// Mitsubishi GX Developer project: Китай гильотина   PLC: FX3U

PROGRAM MAIN
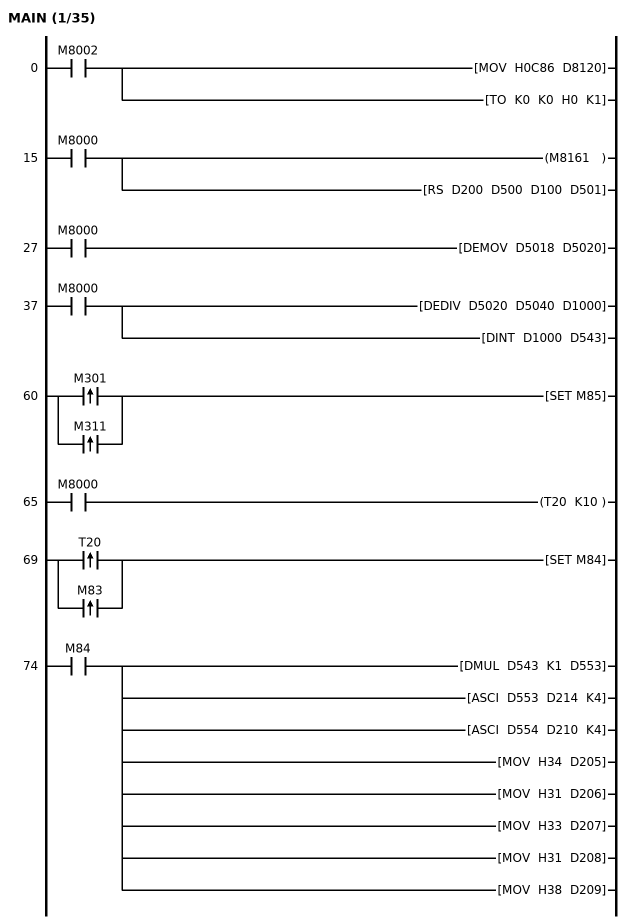
0     LD      M8002
      MOV     H0C86 D8120
      TO      K0 K0 H0 K1
15    LD      M8000
      OUT     M8161
      RS      D200 D500 D100 D501
27    LD      M8000
      DEMOV   D5018 D5020
37    LD      M8000
      DEDIV   D5020 D5040 D1000
      DINT    D1000 D543
60    LDP     M301
      ORP     M311
      SET     M85
65    LD      M8000
      OUT     T20 K10
69    LDP     T20
      ORP     M83
      SET     M84
74    LD      M84
      DMUL    D543 K1 D553
      ASCI    D553 D214 K4
      ASCI    D554 D210 K4
      MOV     H34 D205
      MOV     H31 D206
      MOV     H33 D207
      MOV     H31 D208
      MOV     H38 D209
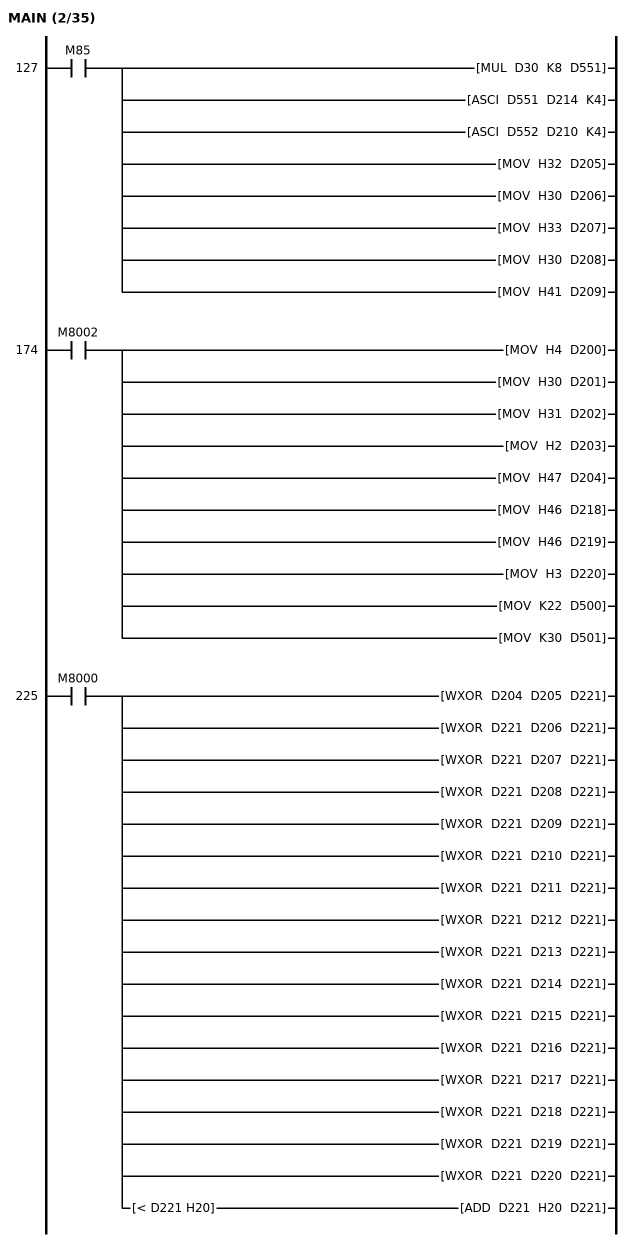
127   LD      M85
      MUL     D30 K8 D551
      ASCI    D551 D214 K4
      ASCI    D552 D210 K4
      MOV     H32 D205
      MOV     H30 D206
      MOV     H33 D207
      MOV     H30 D208
      MOV     H41 D209
174   LD      M8002
      MOV     H4 D200
      MOV     H30 D201
      MOV     H31 D202
      MOV     H2 D203
      MOV     H47 D204
      MOV     H46 D218
      MOV     H46 D219
      MOV     H3 D220
      MOV     K22 D500
      MOV     K30 D501
225   LD      M8000
      WXOR    D204 D205 D221
      WXOR    D221 D206 D221
      WXOR    D221 D207 D221
      WXOR    D221 D208 D221
      WXOR    D221 D209 D221
      WXOR    D221 D210 D221
      WXOR    D221 D211 D221
      WXOR    D221 D212 D221
      WXOR    D221 D213 D221
      WXOR    D221 D214 D221
      WXOR    D221 D215 D221
      WXOR    D221 D216 D221
      WXOR    D221 D217 D221
      WXOR    D221 D218 D221
      WXOR    D221 D219 D221
      WXOR    D221 D220 D221
      AND<    D221 H20
      ADD     D221 H20 D221
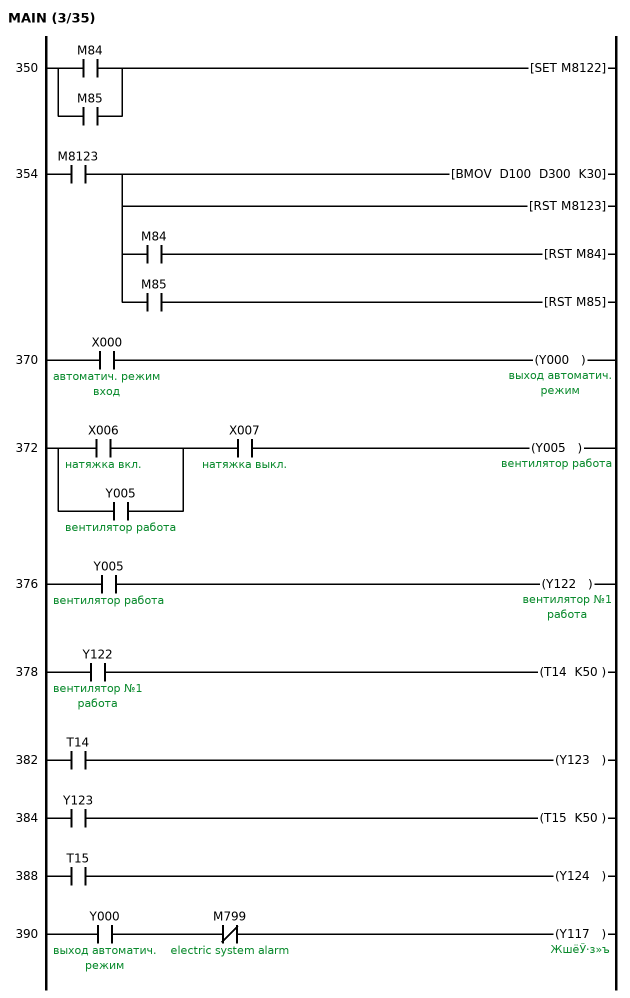
350   LD      M84
      OR      M85
      SET     M8122
354   LD      M8123
      BMOV    D100 D300 K30
      RST     M8123
      MPS
      AND     M84
      RST     M84
      MPP
      AND     M85
      RST     M85
370   LD      X000  ; автоматич. режим вход
      OUT     Y000  ; выход автоматич. режим
372   LD      X006  ; натяжка вкл.
      OR      Y005  ; вентилятор работа
      AND     X007  ; натяжка выкл.
      OUT     Y005  ; вентилятор работа
376   LD      Y005  ; вентилятор работа
      OUT     Y122  ; вентилятор №1 работа
378   LD      Y122  ; вентилятор №1 работа
      OUT     T14 K50
382   LD      T14
      OUT     Y123
384   LD      Y123
      OUT     T15 K50
388   LD      T15
      OUT     Y124
390   LD      Y000  ; выход автоматич. режим
      ANI     M799  ; electric system alarm
      OUT     Y117  ; ЖшёЎ·з»ъ
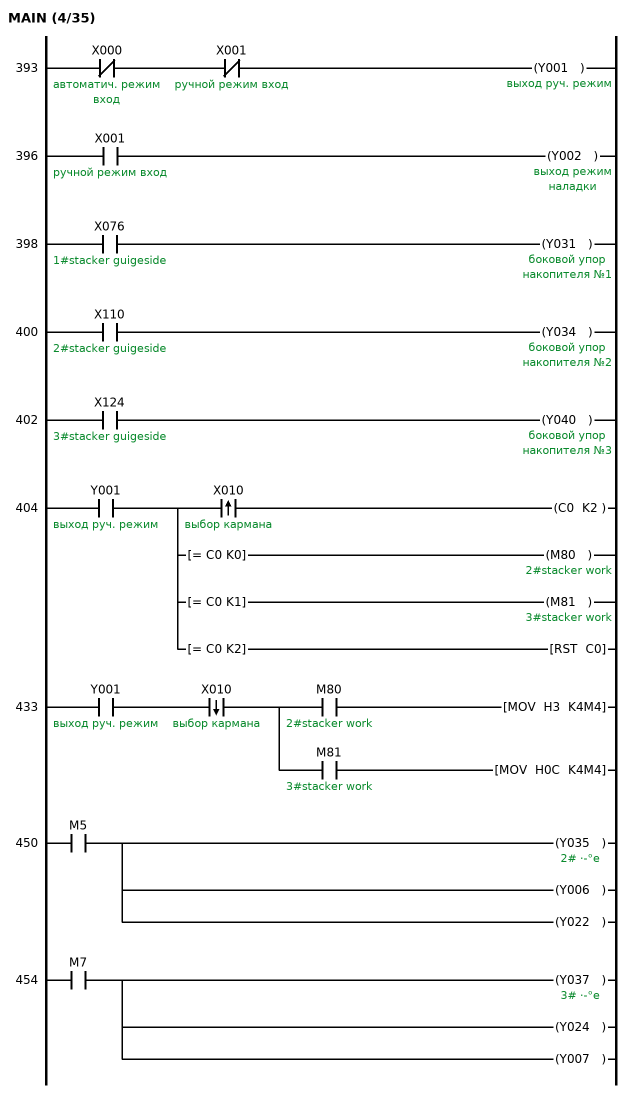
393   LDI     X000  ; автоматич. режим вход
      ANI     X001  ; ручной режим вход
      OUT     Y001  ; выход руч. режим
396   LD      X001  ; ручной режим вход
      OUT     Y002  ; выход режим наладки
398   LD      X076  ; 1#stacker guigeside
      OUT     Y031  ; боковой упор накопителя №1
400   LD      X110  ; 2#stacker guigeside
      OUT     Y034  ; боковой упор накопителя №2
402   LD      X124  ; 3#stacker guigeside
      OUT     Y040  ; боковой упор накопителя №3
404   LD      Y001  ; выход руч. режим
      MPS
      ANDP    X010  ; выбор кармана
      OUT     C0 K2
      MRD
      AND=    C0 K0
      OUT     M80  ; 2#stacker work
      MRD
      AND=    C0 K1
      OUT     M81  ; 3#stacker work
      MPP
      AND=    C0 K2
      RST     C0
433   LD      Y001  ; выход руч. режим
      ANDF    X010  ; выбор кармана
      MPS
      AND     M80  ; 2#stacker work
      MOV     H3 K4M4
      MPP
      AND     M81  ; 3#stacker work
      MOV     H0C K4M4
450   LD      M5
      OUT     Y035  ; 2# ·­°е
      OUT     Y006
      OUT     Y022
454   LD      M7
      OUT     Y037  ; 3# ·­°е
      OUT     Y024
      OUT     Y007
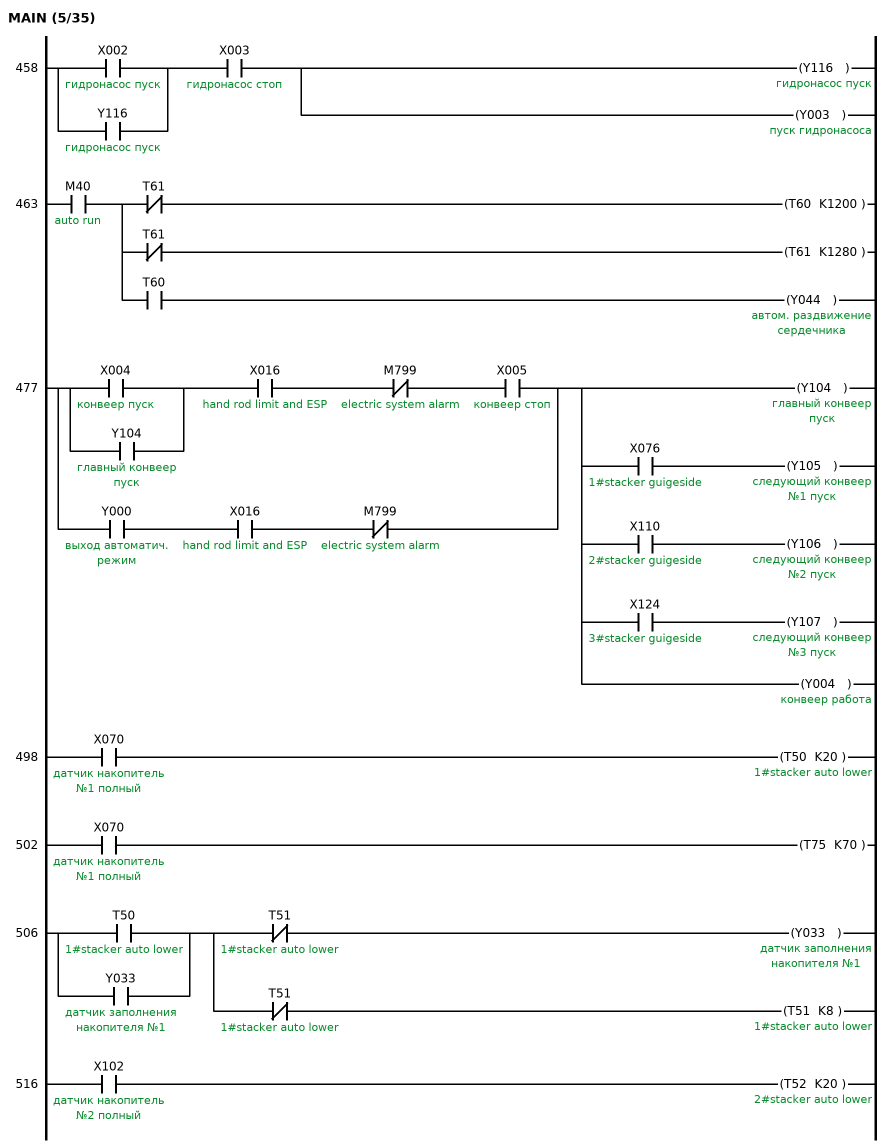
458   LD      X002  ; гидронасос пуск
      OR      Y116  ; гидронасос пуск
      AND     X003  ; гидронасос стоп
      OUT     Y116  ; гидронасос пуск
      OUT     Y003  ; пуск гидронасоса
463   LD      M40  ; auto run
      MPS
      ANI     T61
      OUT     T60 K1200
      MRD
      ANI     T61
      OUT     T61 K1280
      MPP
      AND     T60
      OUT     Y044  ; автом. раздвижение сердечника
477   LD      X004  ; конвеер пуск
      OR      Y104  ; главный конвеер пуск
      AND     X016  ; hand rod limit and ESP
      ANI     M799  ; electric system alarm
      AND     X005  ; конвеер стоп
      LD      Y000  ; выход автоматич. режим
      AND     X016  ; hand rod limit and ESP
      ANI     M799  ; electric system alarm
      ORB
      OUT     Y104  ; главный конвеер пуск
      MPS
      AND     X076  ; 1#stacker guigeside
      OUT     Y105  ; следующий конвеер №1 пуск
      MRD
      AND     X110  ; 2#stacker guigeside
      OUT     Y106  ; следующий конвеер №2 пуск
      MRD
      AND     X124  ; 3#stacker guigeside
      OUT     Y107  ; следующий конвеер №3 пуск
      MPP
      OUT     Y004  ; конвеер работа
498   LD      X070  ; датчик накопитель №1 полный
      OUT     T50 K20  ; 1#stacker auto lower
502   LD      X070  ; датчик накопитель №1 полный
      OUT     T75 K70
506   LD      T50  ; 1#stacker auto lower
      OR      Y033  ; датчик заполнения накопителя №1
      MPS
      ANI     T51  ; 1#stacker auto lower
      OUT     Y033  ; датчик заполнения накопителя №1
      MPP
      ANI     T51  ; 1#stacker auto lower
      OUT     T51 K8  ; 1#stacker auto lower
516   LD      X102  ; датчик накопитель №2 полный
      OUT     T52 K20  ; 2#stacker auto lower
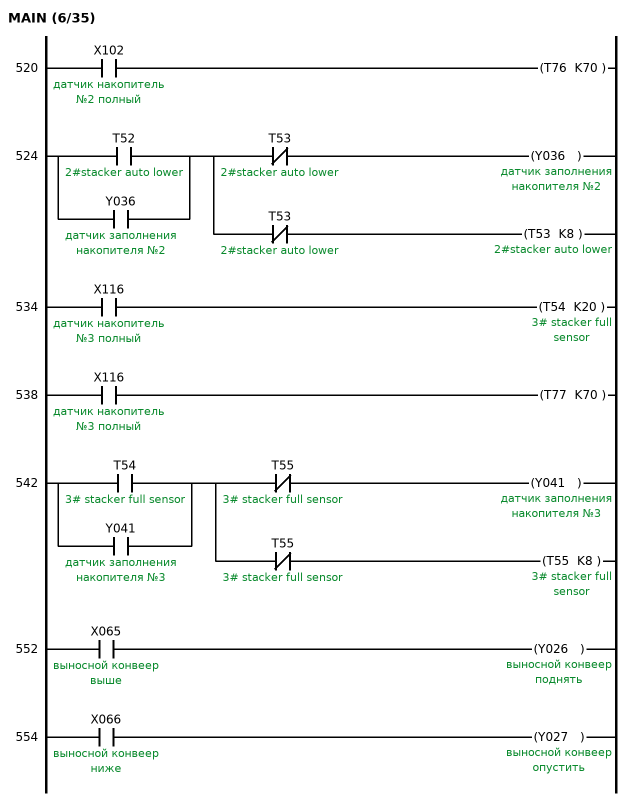
520   LD      X102  ; датчик накопитель №2 полный
      OUT     T76 K70
524   LD      T52  ; 2#stacker auto lower
      OR      Y036  ; датчик заполнения накопителя №2
      MPS
      ANI     T53  ; 2#stacker auto lower
      OUT     Y036  ; датчик заполнения накопителя №2
      MPP
      ANI     T53  ; 2#stacker auto lower
      OUT     T53 K8  ; 2#stacker auto lower
534   LD      X116  ; датчик накопитель №3 полный
      OUT     T54 K20  ; 3# stacker full sensor
538   LD      X116  ; датчик накопитель №3 полный
      OUT     T77 K70
542   LD      T54  ; 3# stacker full sensor
      OR      Y041  ; датчик заполнения накопителя №3
      MPS
      ANI     T55  ; 3# stacker full sensor
      OUT     Y041  ; датчик заполнения накопителя №3
      MPP
      ANI     T55  ; 3# stacker full sensor
      OUT     T55 K8  ; 3# stacker full sensor
552   LD      X065  ; выносной конвеер выше
      OUT     Y026  ; выносной конвеер поднять
554   LD      X066  ; выносной конвеер ниже
      OUT     Y027  ; выносной конвеер опустить
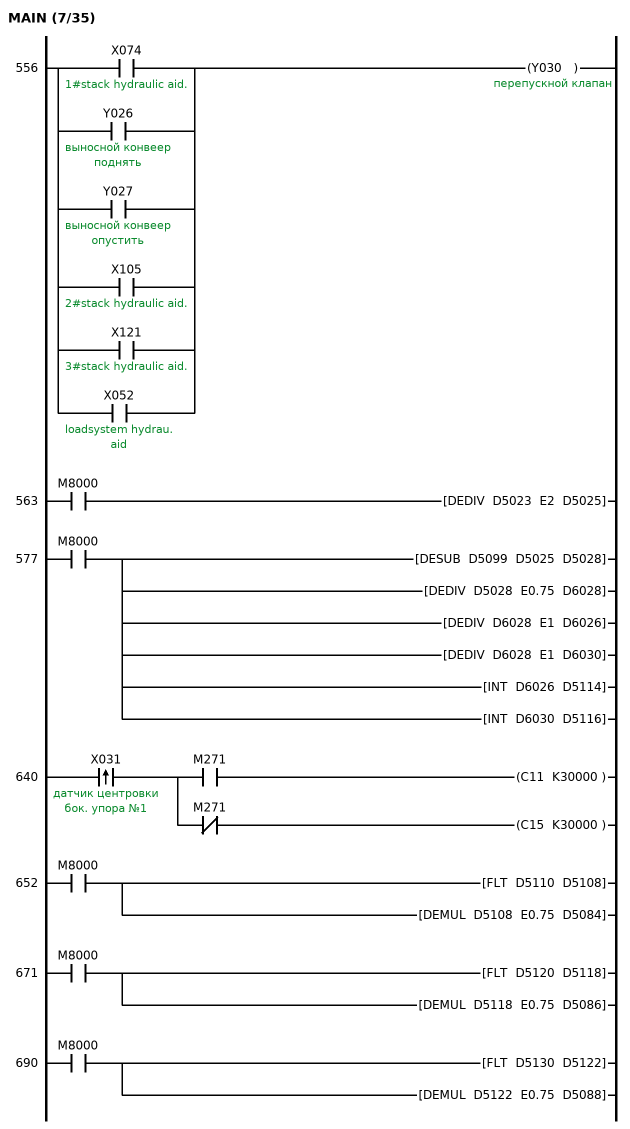
556   LD      X074  ; 1#stack hydraulic aid.
      OR      Y026  ; выносной конвеер поднять
      OR      Y027  ; выносной конвеер опустить
      OR      X105  ; 2#stack hydraulic aid.
      OR      X121  ; 3#stack hydraulic aid.
      OR      X052  ; loadsystem hydrau. aid
      OUT     Y030  ; перепускной клапан
563   LD      M8000
      DEDIV   D5023 E2 D5025
577   LD      M8000
      DESUB   D5099 D5025 D5028
      DEDIV   D5028 E0.75 D6028
      DEDIV   D6028 E1 D6026
      DEDIV   D6028 E1 D6030
      INT     D6026 D5114
      INT     D6030 D5116
640   LDP     X031  ; датчик центровки бок. упора №1
      MPS
      AND     M271
      OUT     C11 K30000
      MPP
      ANI     M271
      OUT     C15 K30000
652   LD      M8000
      FLT     D5110 D5108
      DEMUL   D5108 E0.75 D5084
671   LD      M8000
      FLT     D5120 D5118
      DEMUL   D5118 E0.75 D5086
690   LD      M8000
      FLT     D5130 D5122
      DEMUL   D5122 E0.75 D5088
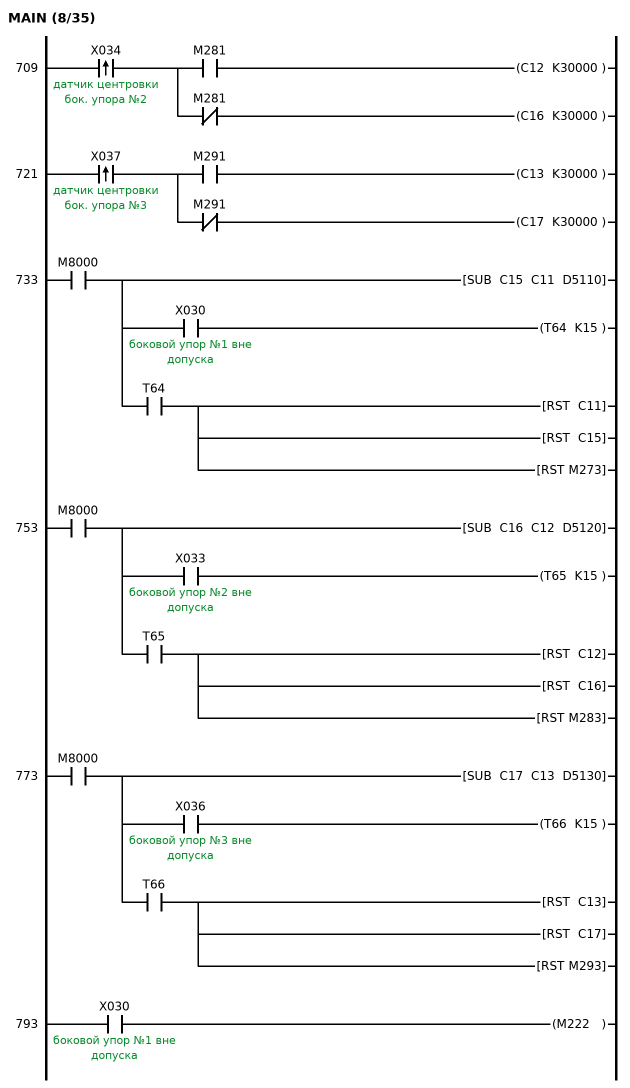
709   LDP     X034  ; датчик центровки бок. упора №2
      MPS
      AND     M281
      OUT     C12 K30000
      MPP
      ANI     M281
      OUT     C16 K30000
721   LDP     X037  ; датчик центровки бок. упора №3
      MPS
      AND     M291
      OUT     C13 K30000
      MPP
      ANI     M291
      OUT     C17 K30000
733   LD      M8000
      SUB     C15 C11 D5110
      MPS
      AND     X030  ; боковой упор №1 вне допуска
      OUT     T64 K15
      MPP
      AND     T64
      RST     C11
      RST     C15
      RST     M273
753   LD      M8000
      SUB     C16 C12 D5120
      MPS
      AND     X033  ; боковой упор №2 вне допуска
      OUT     T65 K15
      MPP
      AND     T65
      RST     C12
      RST     C16
      RST     M283
773   LD      M8000
      SUB     C17 C13 D5130
      MPS
      AND     X036  ; боковой упор №3 вне допуска
      OUT     T66 K15
      MPP
      AND     T66
      RST     C13
      RST     C17
      RST     M293
793   LD      X030  ; боковой упор №1 вне допуска
      OUT     M222
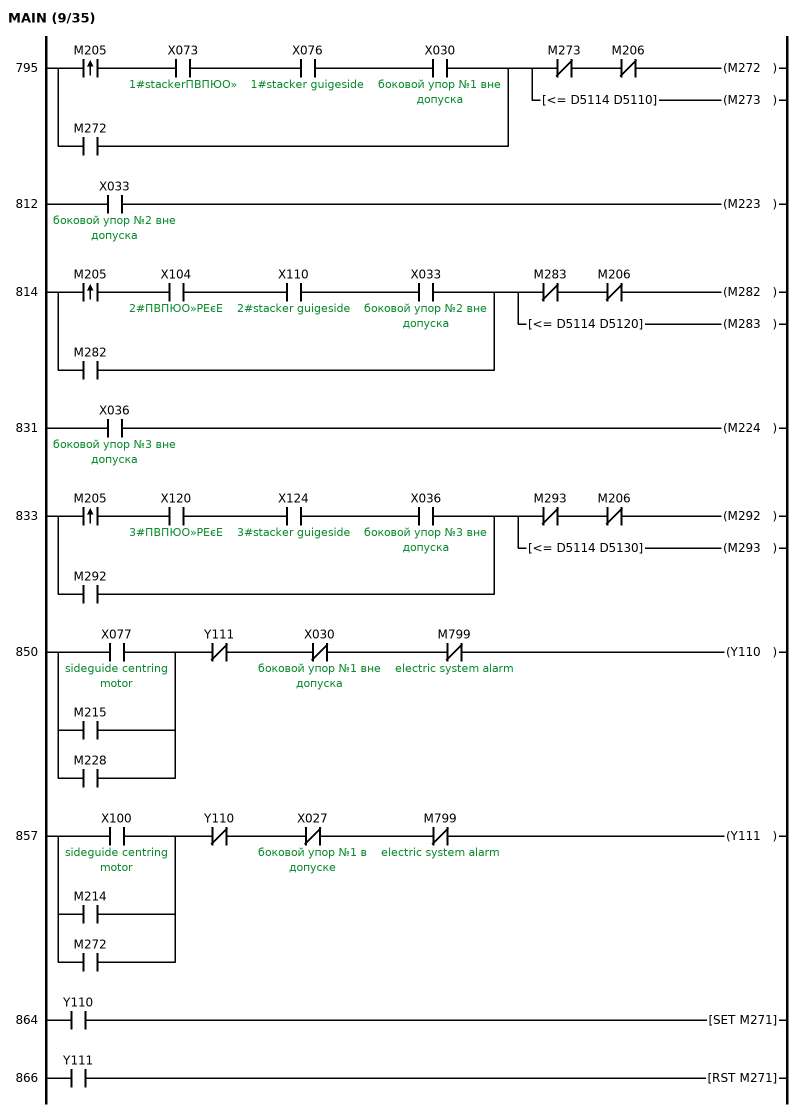
795   LDP     M205
      AND     X073  ; 1#stackerПВПЮО»
      AND     X076  ; 1#stacker guigeside
      AND     X030  ; боковой упор №1 вне допуска
      OR      M272
      MPS
      ANI     M273
      ANI     M206
      OUT     M272
      MPP
      AND<=   D5114 D5110
      OUT     M273
812   LD      X033  ; боковой упор №2 вне допуска
      OUT     M223
814   LDP     M205
      AND     X104  ; 2#ПВПЮО»РЕєЕ
      AND     X110  ; 2#stacker guigeside
      AND     X033  ; боковой упор №2 вне допуска
      OR      M282
      MPS
      ANI     M283
      ANI     M206
      OUT     M282
      MPP
      AND<=   D5114 D5120
      OUT     M283
831   LD      X036  ; боковой упор №3 вне допуска
      OUT     M224
833   LDP     M205
      AND     X120  ; 3#ПВПЮО»РЕєЕ
      AND     X124  ; 3#stacker guigeside
      AND     X036  ; боковой упор №3 вне допуска
      OR      M292
      MPS
      ANI     M293
      ANI     M206
      OUT     M292
      MPP
      AND<=   D5114 D5130
      OUT     M293
850   LD      X077  ; sideguide centring motor
      OR      M215
      OR      M228
      ANI     Y111
      ANI     X030  ; боковой упор №1 вне допуска
      ANI     M799  ; electric system alarm
      OUT     Y110
857   LD      X100  ; sideguide centring motor
      OR      M214
      OR      M272
      ANI     Y110
      ANI     X027  ; боковой упор №1 в допуске
      ANI     M799  ; electric system alarm
      OUT     Y111
864   LD      Y110
      SET     M271
866   LD      Y111
      RST     M271
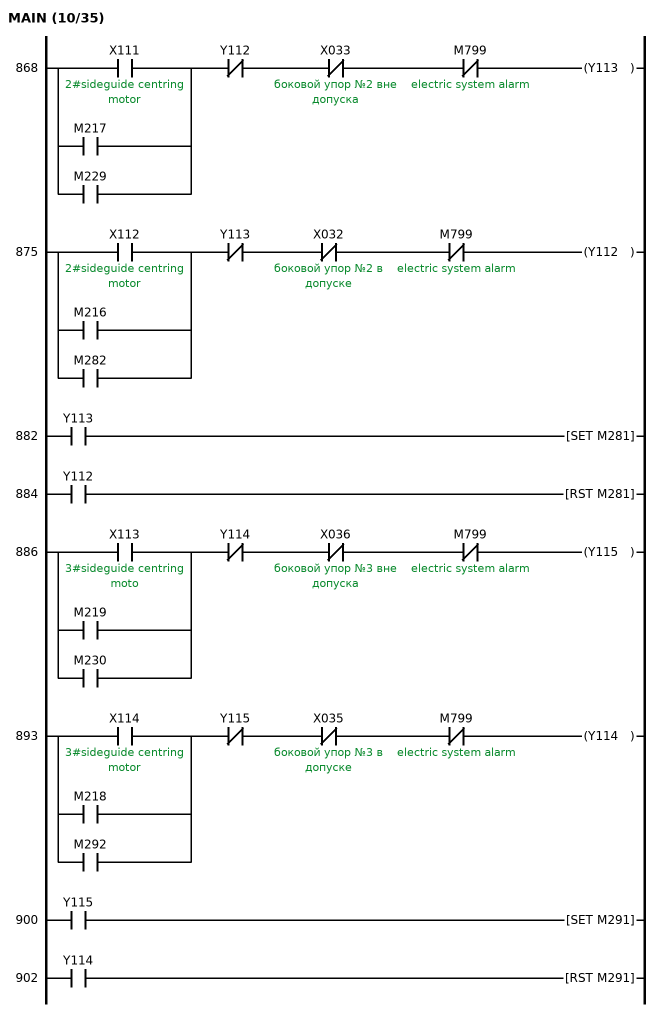
868   LD      X111  ; 2#sideguide centring motor
      OR      M217
      OR      M229
      ANI     Y112
      ANI     X033  ; боковой упор №2 вне допуска
      ANI     M799  ; electric system alarm
      OUT     Y113
875   LD      X112  ; 2#sideguide centring motor
      OR      M216
      OR      M282
      ANI     Y113
      ANI     X032  ; боковой упор №2 в допуске
      ANI     M799  ; electric system alarm
      OUT     Y112
882   LD      Y113
      SET     M281
884   LD      Y112
      RST     M281
886   LD      X113  ; 3#sideguide centring moto
      OR      M219
      OR      M230
      ANI     Y114
      ANI     X036  ; боковой упор №3 вне допуска
      ANI     M799  ; electric system alarm
      OUT     Y115
893   LD      X114  ; 3#sideguide centring motor
      OR      M218
      OR      M292
      ANI     Y115
      ANI     X035  ; боковой упор №3 в допуске
      ANI     M799  ; electric system alarm
      OUT     Y114
900   LD      Y115
      SET     M291
902   LD      Y114
      RST     M291
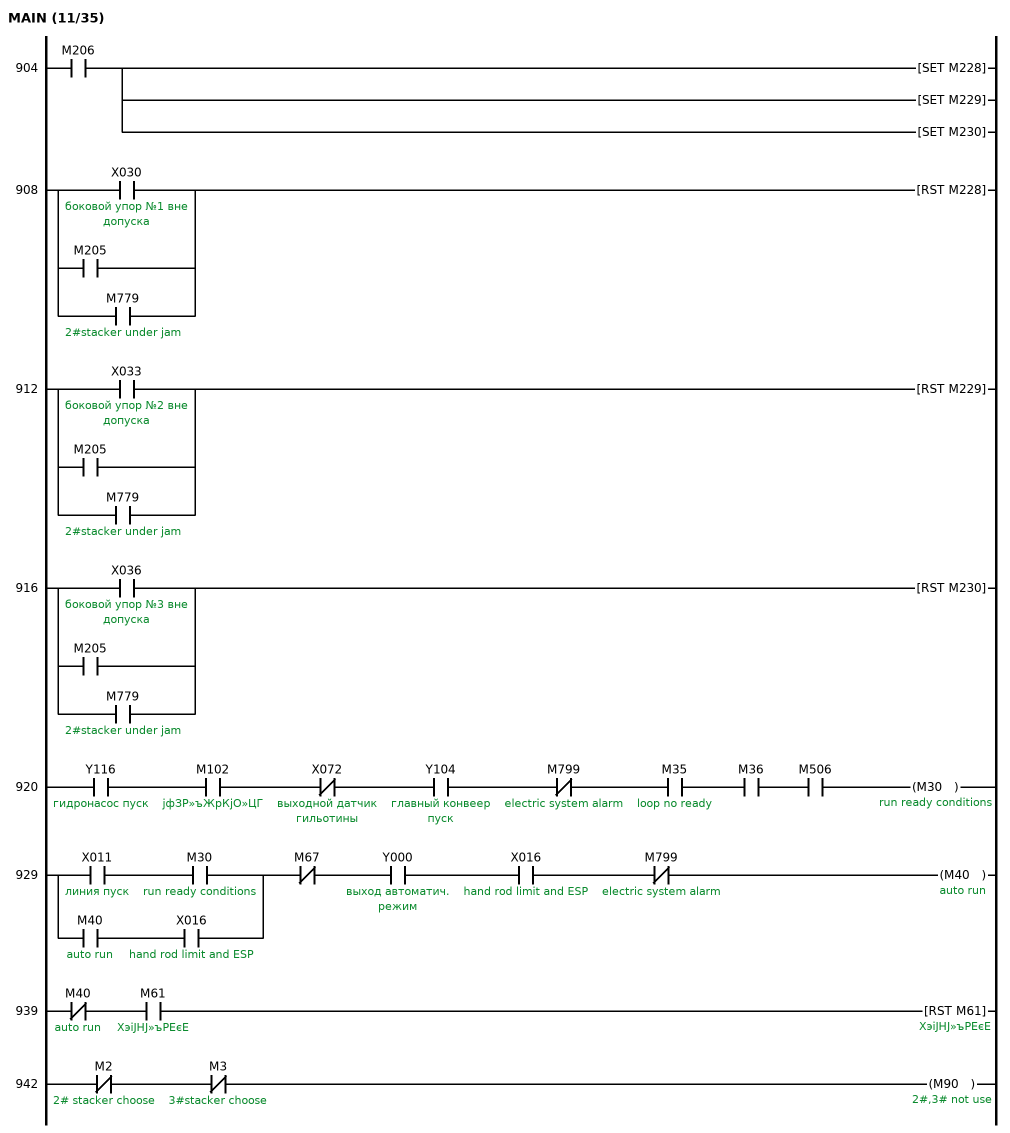
904   LD      M206
      SET     M228
      SET     M229
      SET     M230
908   LD      X030  ; боковой упор №1 вне допуска
      OR      M205
      OR      M779  ; 2#stacker under jam
      RST     M228
912   LD      X033  ; боковой упор №2 вне допуска
      OR      M205
      OR      M779  ; 2#stacker under jam
      RST     M229
916   LD      X036  ; боковой упор №3 вне допуска
      OR      M205
      OR      M779  ; 2#stacker under jam
      RST     M230
920   LD      Y116  ; гидронасос пуск
      AND     M102  ; јфЗР»ъЖрКјО»ЦГ
      ANI     X072  ; выходной датчик гильотины
      AND     Y104  ; главный конвеер пуск
      ANI     M799  ; electric system alarm
      AND     M35  ; loop no ready
      AND     M36
      AND     M506
      OUT     M30  ; run ready conditions
929   LD      X011  ; линия пуск
      AND     M30  ; run ready conditions
      LD      M40  ; auto run
      AND     X016  ; hand rod limit and ESP
      ORB
      ANI     M67
      AND     Y000  ; выход автоматич. режим
      AND     X016  ; hand rod limit and ESP
      ANI     M799  ; electric system alarm
      OUT     M40  ; auto run
939   LDI     M40  ; auto run
      AND     M61  ; ХэіЈНЈ»ъРЕєЕ
      RST     M61  ; ХэіЈНЈ»ъРЕєЕ
942   LDI     M2  ; 2# stacker choose
      ANI     M3  ; 3#stacker choose
      OUT     M90  ; 2#,3# not use
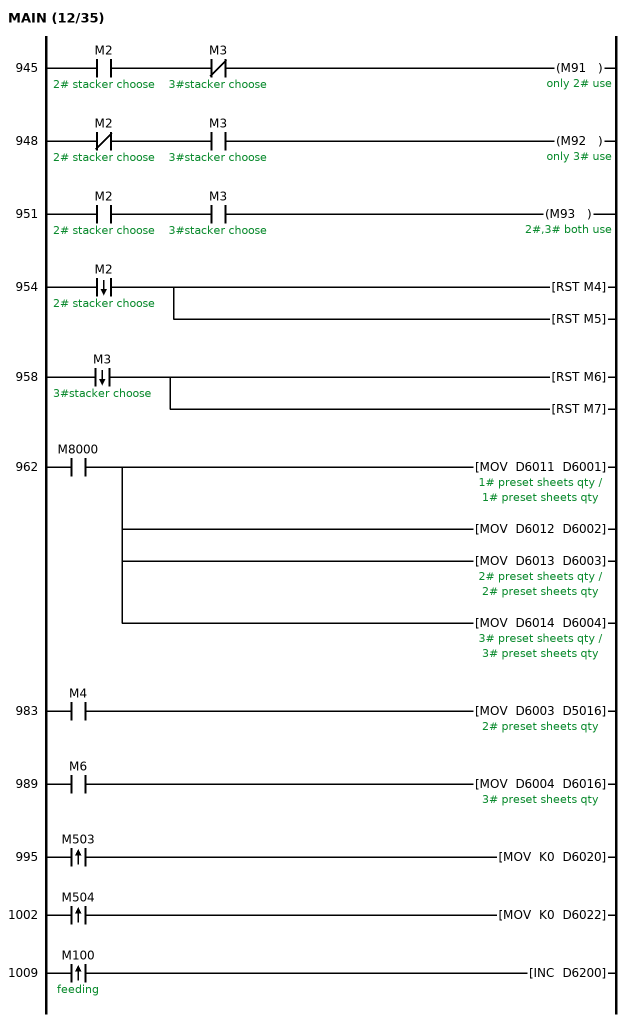
945   LD      M2  ; 2# stacker choose
      ANI     M3  ; 3#stacker choose
      OUT     M91  ; only 2# use
948   LDI     M2  ; 2# stacker choose
      AND     M3  ; 3#stacker choose
      OUT     M92  ; only 3# use
951   LD      M2  ; 2# stacker choose
      AND     M3  ; 3#stacker choose
      OUT     M93  ; 2#,3# both use
954   LDF     M2  ; 2# stacker choose
      RST     M4
      RST     M5
958   LDF     M3  ; 3#stacker choose
      RST     M6
      RST     M7
962   LD      M8000
      MOV     D6011 D6001  ; 1# preset sheets qty / 1# preset sheets qty
      MOV     D6012 D6002
      MOV     D6013 D6003  ; 2# preset sheets qty / 2# preset sheets qty
      MOV     D6014 D6004  ; 3# preset sheets qty / 3# preset sheets qty
983   LD      M4
      MOV     D6003 D5016
989   LD      M6
      MOV     D6004 D6016
995   LDP     M503
      MOV     K0 D6020
1002  LDP     M504
      MOV     K0 D6022
1009  LDP     M100  ; feeding
      INC     D6200
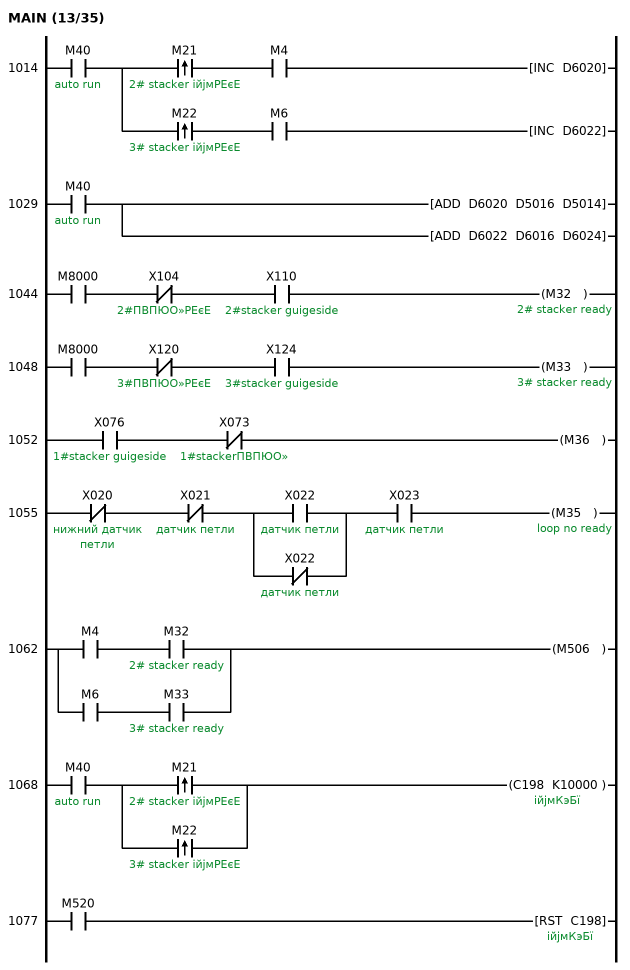
1014  LD      M40  ; auto run
      MPS
      ANDP    M21  ; 2# stacker ійјмРЕєЕ
      AND     M4
      INC     D6020
      MPP
      ANDP    M22  ; 3# stacker ійјмРЕєЕ
      AND     M6
      INC     D6022
1029  LD      M40  ; auto run
      ADD     D6020 D5016 D5014
      ADD     D6022 D6016 D6024
1044  LD      M8000
      ANI     X104  ; 2#ПВПЮО»РЕєЕ
      AND     X110  ; 2#stacker guigeside
      OUT     M32  ; 2# stacker ready
1048  LD      M8000
      ANI     X120  ; 3#ПВПЮО»РЕєЕ
      AND     X124  ; 3#stacker guigeside
      OUT     M33  ; 3# stacker ready
1052  LD      X076  ; 1#stacker guigeside
      ANI     X073  ; 1#stackerПВПЮО»
      OUT     M36
1055  LDI     X020  ; нижний датчик петли
      ANI     X021  ; датчик петли
      LD      X022  ; датчик петли
      ORI     X022  ; датчик петли
      ANB
      AND     X023  ; датчик петли
      OUT     M35  ; loop no ready
1062  LD      M4
      AND     M32  ; 2# stacker ready
      LD      M6
      AND     M33  ; 3# stacker ready
      ORB
      OUT     M506
1068  LD      M40  ; auto run
      LDP     M21  ; 2# stacker ійјмРЕєЕ
      ORP     M22  ; 3# stacker ійјмРЕєЕ
      ANB
      OUT     C198 K10000  ; ійјмКэБї
1077  LD      M520
      RST     C198  ; ійјмКэБї
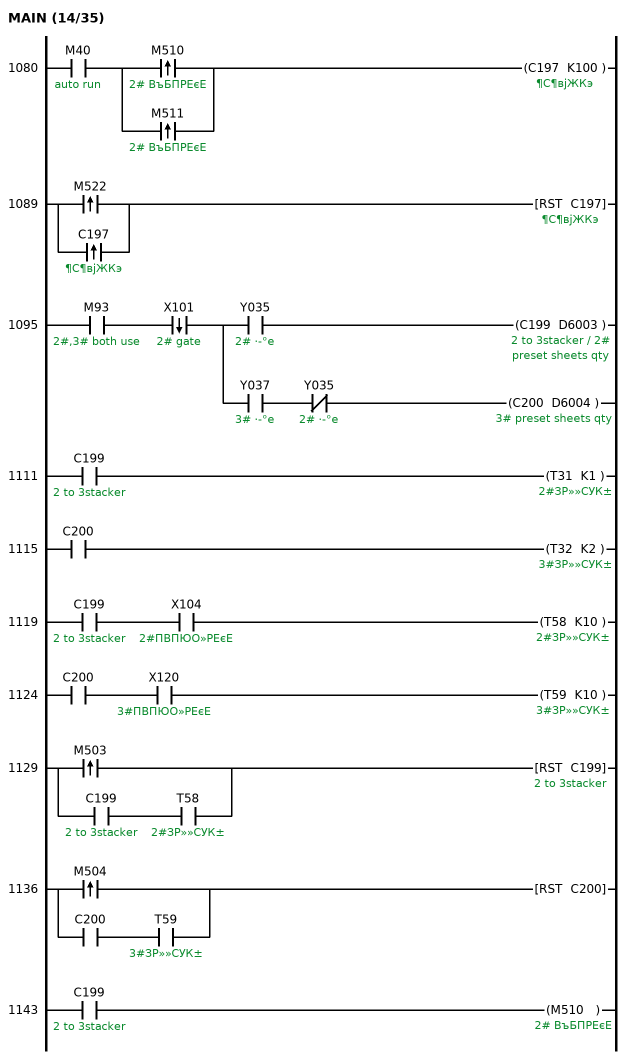
1080  LD      M40  ; auto run
      LDP     M510  ; 2# ВъБПРЕєЕ
      ORP     M511  ; 2# ВъБПРЕєЕ
      ANB
      OUT     C197 K100  ; ¶С¶вјЖКэ
1089  LDP     M522
      ORP     C197  ; ¶С¶вјЖКэ
      RST     C197  ; ¶С¶вјЖКэ
1095  LD      M93  ; 2#,3# both use
      ANDF    X101  ; 2# gate
      MPS
      AND     Y035  ; 2# ·­°е
      OUT     C199 D6003  ; 2 to 3stacker / 2# preset sheets qty
      MPP
      AND     Y037  ; 3# ·­°е
      ANI     Y035  ; 2# ·­°е
      OUT     C200 D6004  ; 3# preset sheets qty
1111  LD      C199  ; 2 to 3stacker
      OUT     T31 K1  ; 2#ЗР»»СУК±
1115  LD      C200
      OUT     T32 K2  ; 3#ЗР»»СУК±
1119  LD      C199  ; 2 to 3stacker
      AND     X104  ; 2#ПВПЮО»РЕєЕ
      OUT     T58 K10  ; 2#ЗР»»СУК±
1124  LD      C200
      AND     X120  ; 3#ПВПЮО»РЕєЕ
      OUT     T59 K10  ; 3#ЗР»»СУК±
1129  LDP     M503
      LD      C199  ; 2 to 3stacker
      AND     T58  ; 2#ЗР»»СУК±
      ORB
      RST     C199  ; 2 to 3stacker
1136  LDP     M504
      LD      C200
      AND     T59  ; 3#ЗР»»СУК±
      ORB
      RST     C200
1143  LD      C199  ; 2 to 3stacker
      OUT     M510  ; 2# ВъБПРЕєЕ
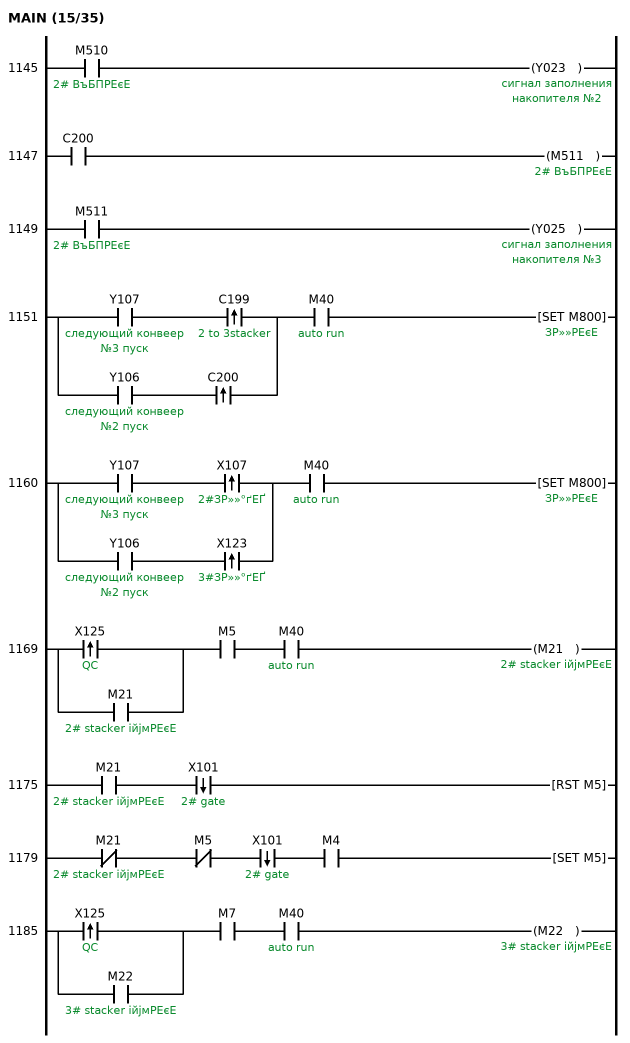
1145  LD      M510  ; 2# ВъБПРЕєЕ
      OUT     Y023  ; сигнал заполнения накопителя №2
1147  LD      C200
      OUT     M511  ; 2# ВъБПРЕєЕ
1149  LD      M511  ; 2# ВъБПРЕєЕ
      OUT     Y025  ; сигнал заполнения накопителя №3
1151  LD      Y107  ; следующий конвеер №3 пуск
      ANDP    C199  ; 2 to 3stacker
      LD      Y106  ; следующий конвеер №2 пуск
      ANDP    C200
      ORB
      AND     M40  ; auto run
      SET     M800  ; ЗР»»РЕєЕ
1160  LD      Y107  ; следующий конвеер №3 пуск
      ANDP    X107  ; 2#ЗР»»°ґЕҐ
      LD      Y106  ; следующий конвеер №2 пуск
      ANDP    X123  ; 3#ЗР»»°ґЕҐ
      ORB
      AND     M40  ; auto run
      SET     M800  ; ЗР»»РЕєЕ
1169  LDP     X125  ; QC
      OR      M21  ; 2# stacker ійјмРЕєЕ
      AND     M5
      AND     M40  ; auto run
      OUT     M21  ; 2# stacker ійјмРЕєЕ
1175  LD      M21  ; 2# stacker ійјмРЕєЕ
      ANDF    X101  ; 2# gate
      RST     M5
1179  LDI     M21  ; 2# stacker ійјмРЕєЕ
      ANI     M5
      ANDF    X101  ; 2# gate
      AND     M4
      SET     M5
1185  LDP     X125  ; QC
      OR      M22  ; 3# stacker ійјмРЕєЕ
      AND     M7
      AND     M40  ; auto run
      OUT     M22  ; 3# stacker ійјмРЕєЕ
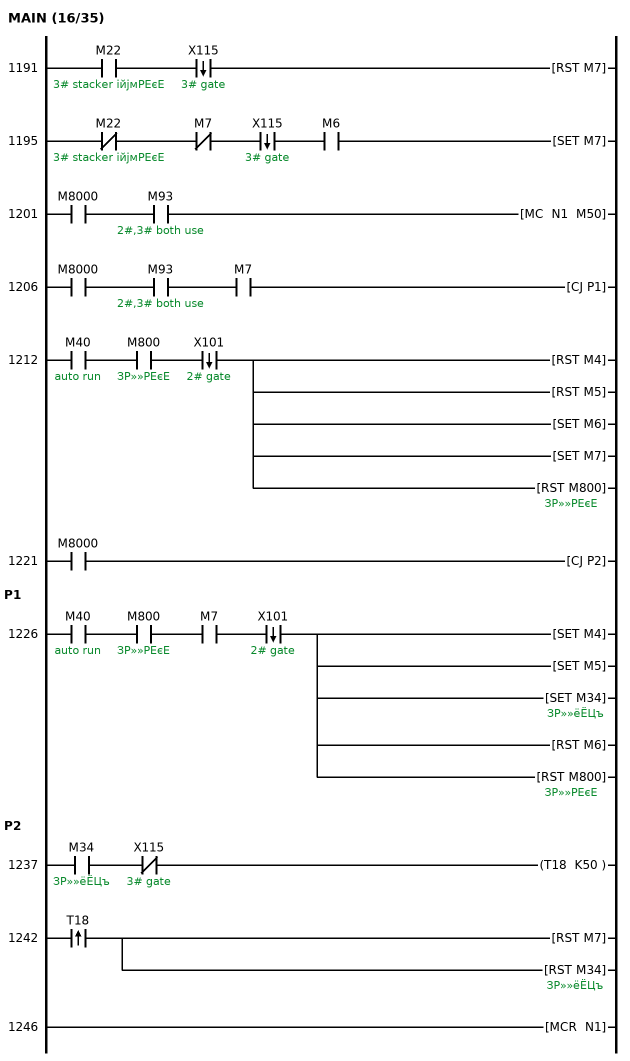
1191  LD      M22  ; 3# stacker ійјмРЕєЕ
      ANDF    X115  ; 3# gate
      RST     M7
1195  LDI     M22  ; 3# stacker ійјмРЕєЕ
      ANI     M7
      ANDF    X115  ; 3# gate
      AND     M6
      SET     M7
1201  LD      M8000
      AND     M93  ; 2#,3# both use
      MC      N1 M50
1206  LD      M8000
      AND     M93  ; 2#,3# both use
      AND     M7
      CJ      P1
1212  LD      M40  ; auto run
      AND     M800  ; ЗР»»РЕєЕ
      ANDF    X101  ; 2# gate
      RST     M4
      RST     M5
      SET     M6
      SET     M7
      RST     M800  ; ЗР»»РЕєЕ
1221  LD      M8000
      CJ      P2
      P1
1226  LD      M40  ; auto run
      AND     M800  ; ЗР»»РЕєЕ
      AND     M7
      ANDF    X101  ; 2# gate
      SET     M4
      SET     M5
      SET     M34  ; ЗР»»ёЁЦъ
      RST     M6
      RST     M800  ; ЗР»»РЕєЕ
      P2
1237  LD      M34  ; ЗР»»ёЁЦъ
      ANI     X115  ; 3# gate
      OUT     T18 K50
1242  LDP     T18
      RST     M7
      RST     M34  ; ЗР»»ёЁЦъ
1246  MCR     N1
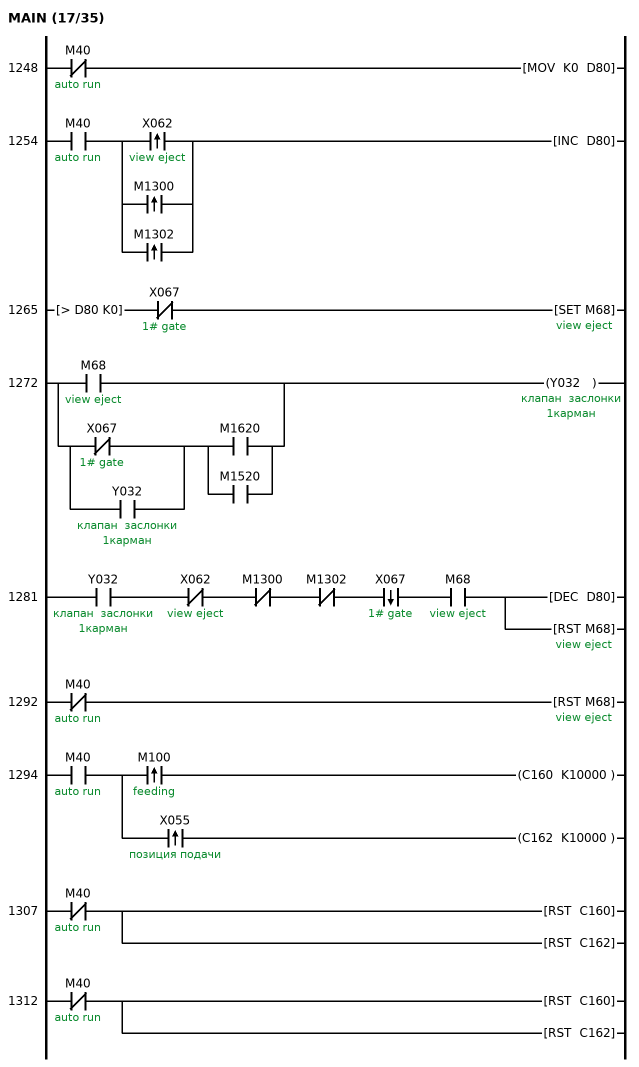
1248  LDI     M40  ; auto run
      MOV     K0 D80
1254  LD      M40  ; auto run
      LDP     X062  ; view eject
      ORP     M1300
      ORP     M1302
      ANB
      INC     D80
1265  LD>     D80 K0
      ANI     X067  ; 1# gate
      SET     M68  ; view eject
1272  LD      M68  ; view eject
      LDI     X067  ; 1# gate
      OR      Y032  ; клапан  заслонки 1карман
      LD      M1620
      OR      M1520
      ANB
      ORB
      OUT     Y032  ; клапан  заслонки 1карман
1281  LD      Y032  ; клапан  заслонки 1карман
      ANI     X062  ; view eject
      ANI     M1300
      ANI     M1302
      ANDF    X067  ; 1# gate
      AND     M68  ; view eject
      DEC     D80
      RST     M68  ; view eject
1292  LDI     M40  ; auto run
      RST     M68  ; view eject
1294  LD      M40  ; auto run
      MPS
      ANDP    M100  ; feeding
      OUT     C160 K10000
      MPP
      ANDP    X055  ; позиция подачи
      OUT     C162 K10000
1307  LDI     M40  ; auto run
      RST     C160
      RST     C162
1312  LDI     M40  ; auto run
      RST     C160
      RST     C162
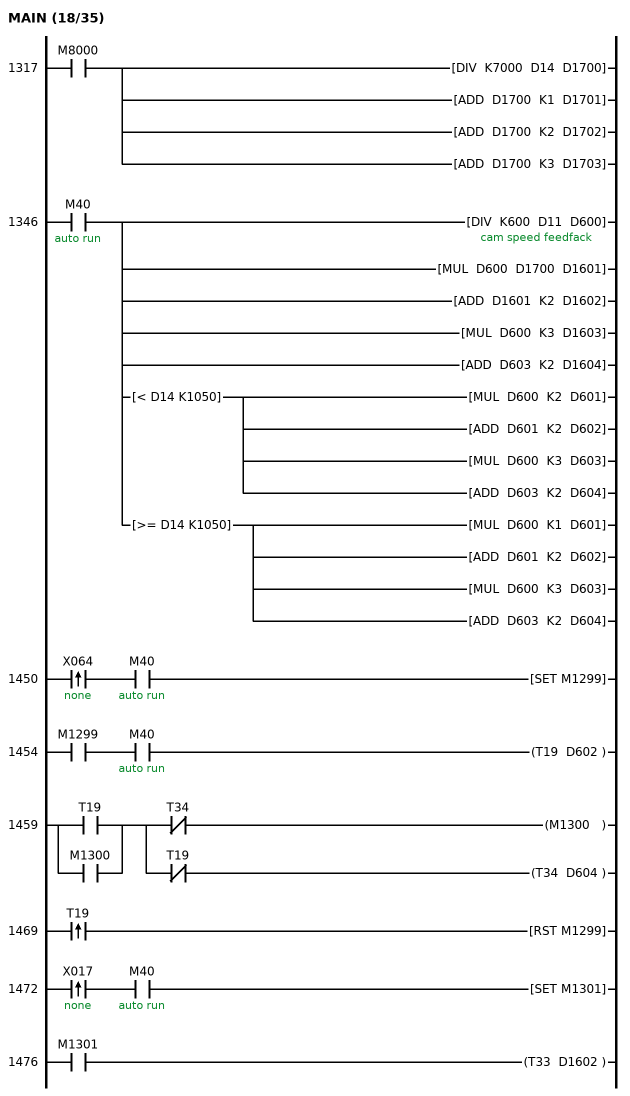
1317  LD      M8000
      DIV     K7000 D14 D1700
      ADD     D1700 K1 D1701
      ADD     D1700 K2 D1702
      ADD     D1700 K3 D1703
1346  LD      M40  ; auto run
      DIV     K600 D11 D600  ; cam speed feedfack
      MUL     D600 D1700 D1601
      ADD     D1601 K2 D1602
      MUL     D600 K3 D1603
      ADD     D603 K2 D1604
      MPS
      AND<    D14 K1050
      MUL     D600 K2 D601
      ADD     D601 K2 D602
      MUL     D600 K3 D603
      ADD     D603 K2 D604
      MPP
      AND>=   D14 K1050
      MUL     D600 K1 D601
      ADD     D601 K2 D602
      MUL     D600 K3 D603
      ADD     D603 K2 D604
1450  LDP     X064  ; none
      AND     M40  ; auto run
      SET     M1299
1454  LD      M1299
      AND     M40  ; auto run
      OUT     T19 D602
1459  LD      T19
      OR      M1300
      MPS
      ANI     T34
      OUT     M1300
      MPP
      ANI     T19
      OUT     T34 D604
1469  LDP     T19
      RST     M1299
1472  LDP     X017  ; none
      AND     M40  ; auto run
      SET     M1301
1476  LD      M1301
      OUT     T33 D1602
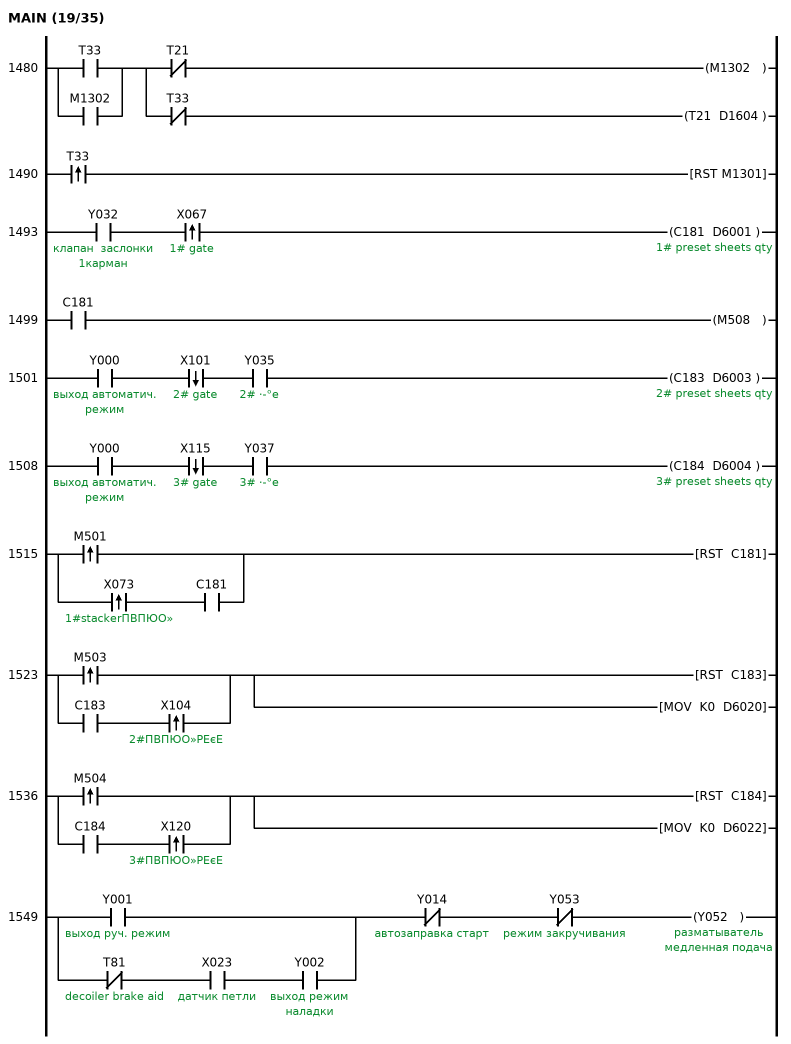
1480  LD      T33
      OR      M1302
      MPS
      ANI     T21
      OUT     M1302
      MPP
      ANI     T33
      OUT     T21 D1604
1490  LDP     T33
      RST     M1301
1493  LD      Y032  ; клапан  заслонки 1карман
      ANDP    X067  ; 1# gate
      OUT     C181 D6001  ; 1# preset sheets qty
1499  LD      C181
      OUT     M508
1501  LD      Y000  ; выход автоматич. режим
      ANDF    X101  ; 2# gate
      AND     Y035  ; 2# ·­°е
      OUT     C183 D6003  ; 2# preset sheets qty
1508  LD      Y000  ; выход автоматич. режим
      ANDF    X115  ; 3# gate
      AND     Y037  ; 3# ·­°е
      OUT     C184 D6004  ; 3# preset sheets qty
1515  LDP     M501
      LDP     X073  ; 1#stackerПВПЮО»
      AND     C181
      ORB
      RST     C181
1523  LDP     M503
      LD      C183
      ANDP    X104  ; 2#ПВПЮО»РЕєЕ
      ORB
      RST     C183
      MOV     K0 D6020
1536  LDP     M504
      LD      C184
      ANDP    X120  ; 3#ПВПЮО»РЕєЕ
      ORB
      RST     C184
      MOV     K0 D6022
1549  LD      Y001  ; выход руч. режим
      LDI     T81  ; decoiler brake aid
      AND     X023  ; датчик петли
      AND     Y002  ; выход режим наладки
      ORB
      ANI     Y014  ; автозаправка старт
      ANI     Y053  ; режим закручивания
      OUT     Y052  ; разматыватель медленная подача
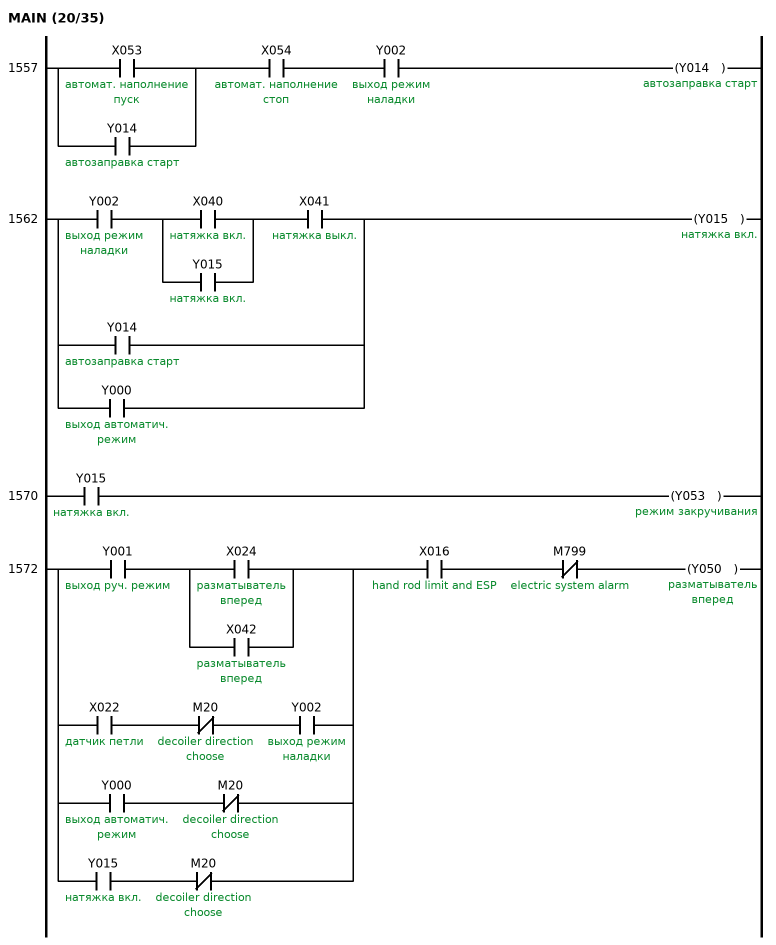
1557  LD      X053  ; автомат. наполнение пуск
      OR      Y014  ; автозаправка старт
      AND     X054  ; автомат. наполнение стоп
      AND     Y002  ; выход режим наладки
      OUT     Y014  ; автозаправка старт
1562  LD      Y002  ; выход режим наладки
      LD      X040  ; натяжка вкл.
      OR      Y015  ; натяжка вкл.
      ANB
      AND     X041  ; натяжка выкл.
      OR      Y014  ; автозаправка старт
      OR      Y000  ; выход автоматич. режим
      OUT     Y015  ; натяжка вкл.
1570  LD      Y015  ; натяжка вкл.
      OUT     Y053  ; режим закручивания
1572  LD      Y001  ; выход руч. режим
      LD      X024  ; разматыватель вперед
      OR      X042  ; разматыватель вперед
      ANB
      LD      X022  ; датчик петли
      ANI     M20  ; decoiler direction choose
      AND     Y002  ; выход режим наладки
      ORB
      LD      Y000  ; выход автоматич. режим
      ANI     M20  ; decoiler direction choose
      ORB
      LD      Y015  ; натяжка вкл.
      ANI     M20  ; decoiler direction choose
      ORB
      AND     X016  ; hand rod limit and ESP
      ANI     M799  ; electric system alarm
      OUT     Y050  ; разматыватель вперед
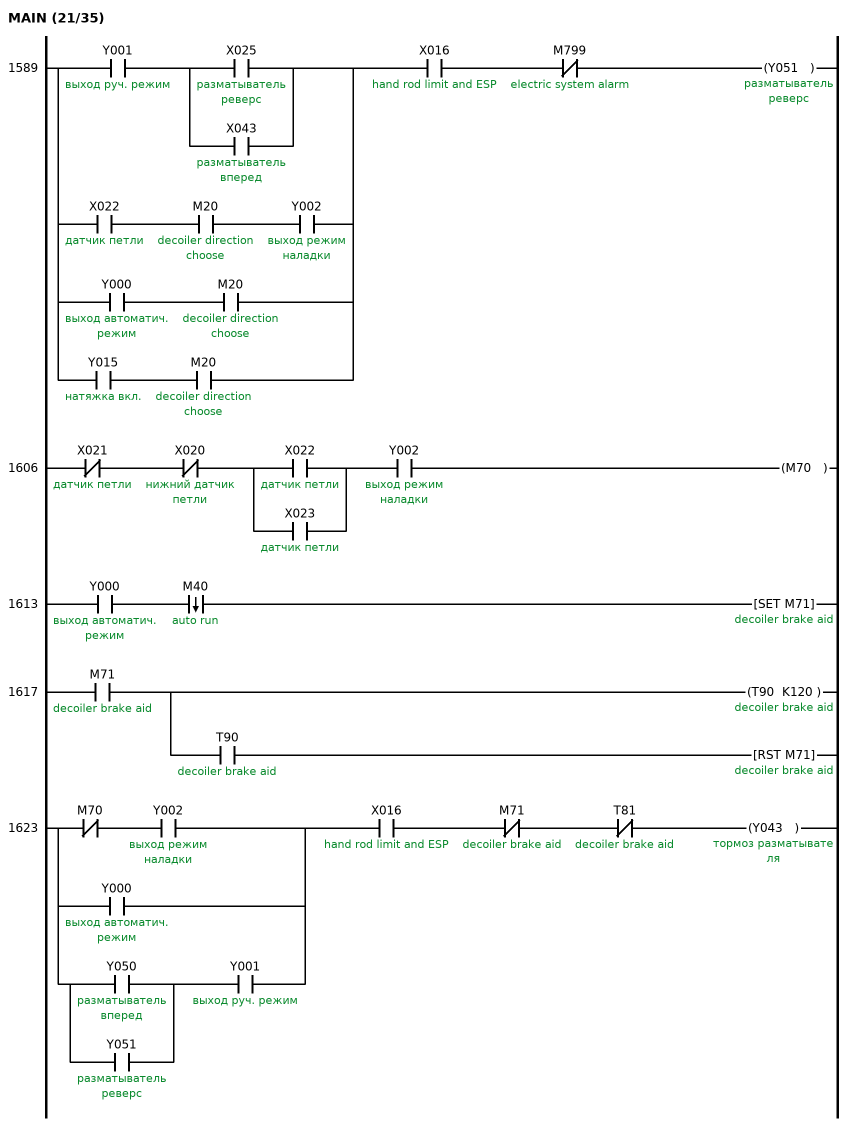
1589  LD      Y001  ; выход руч. режим
      LD      X025  ; разматыватель реверс
      OR      X043  ; разматыватель вперед
      ANB
      LD      X022  ; датчик петли
      AND     M20  ; decoiler direction choose
      AND     Y002  ; выход режим наладки
      ORB
      LD      Y000  ; выход автоматич. режим
      AND     M20  ; decoiler direction choose
      ORB
      LD      Y015  ; натяжка вкл.
      AND     M20  ; decoiler direction choose
      ORB
      AND     X016  ; hand rod limit and ESP
      ANI     M799  ; electric system alarm
      OUT     Y051  ; разматыватель реверс
1606  LDI     X021  ; датчик петли
      ANI     X020  ; нижний датчик петли
      LD      X022  ; датчик петли
      OR      X023  ; датчик петли
      ANB
      AND     Y002  ; выход режим наладки
      OUT     M70
1613  LD      Y000  ; выход автоматич. режим
      ANDF    M40  ; auto run
      SET     M71  ; decoiler brake aid
1617  LD      M71  ; decoiler brake aid
      OUT     T90 K120  ; decoiler brake aid
      AND     T90  ; decoiler brake aid
      RST     M71  ; decoiler brake aid
1623  LDI     M70
      AND     Y002  ; выход режим наладки
      OR      Y000  ; выход автоматич. режим
      LD      Y050  ; разматыватель вперед
      OR      Y051  ; разматыватель реверс
      AND     Y001  ; выход руч. режим
      ORB
      AND     X016  ; hand rod limit and ESP
      ANI     M71  ; decoiler brake aid
      ANI     T81  ; decoiler brake aid
      OUT     Y043  ; тормоз разматывателя
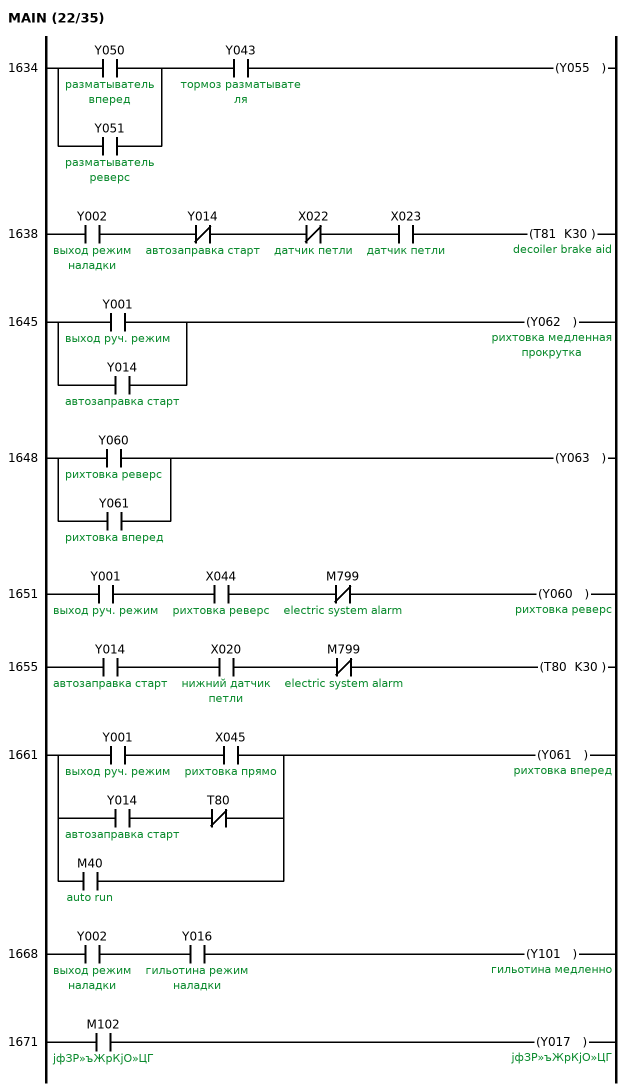
1634  LD      Y050  ; разматыватель вперед
      OR      Y051  ; разматыватель реверс
      AND     Y043  ; тормоз разматывателя
      OUT     Y055
1638  LD      Y002  ; выход режим наладки
      ANI     Y014  ; автозаправка старт
      ANI     X022  ; датчик петли
      AND     X023  ; датчик петли
      OUT     T81 K30  ; decoiler brake aid
1645  LD      Y001  ; выход руч. режим
      OR      Y014  ; автозаправка старт
      OUT     Y062  ; рихтовка медленная прокрутка
1648  LD      Y060  ; рихтовка реверс
      OR      Y061  ; рихтовка вперед
      OUT     Y063
1651  LD      Y001  ; выход руч. режим
      AND     X044  ; рихтовка реверс
      ANI     M799  ; electric system alarm
      OUT     Y060  ; рихтовка реверс
1655  LD      Y014  ; автозаправка старт
      AND     X020  ; нижний датчик петли
      ANI     M799  ; electric system alarm
      OUT     T80 K30
1661  LD      Y001  ; выход руч. режим
      AND     X045  ; рихтовка прямо
      LD      Y014  ; автозаправка старт
      ANI     T80
      ORB
      OR      M40  ; auto run
      OUT     Y061  ; рихтовка вперед
1668  LD      Y002  ; выход режим наладки
      AND     Y016  ; гильотина режим наладки
      OUT     Y101  ; гильотина медленно
1671  LD      M102  ; јфЗР»ъЖрКјО»ЦГ
      OUT     Y017  ; јфЗР»ъЖрКјО»ЦГ
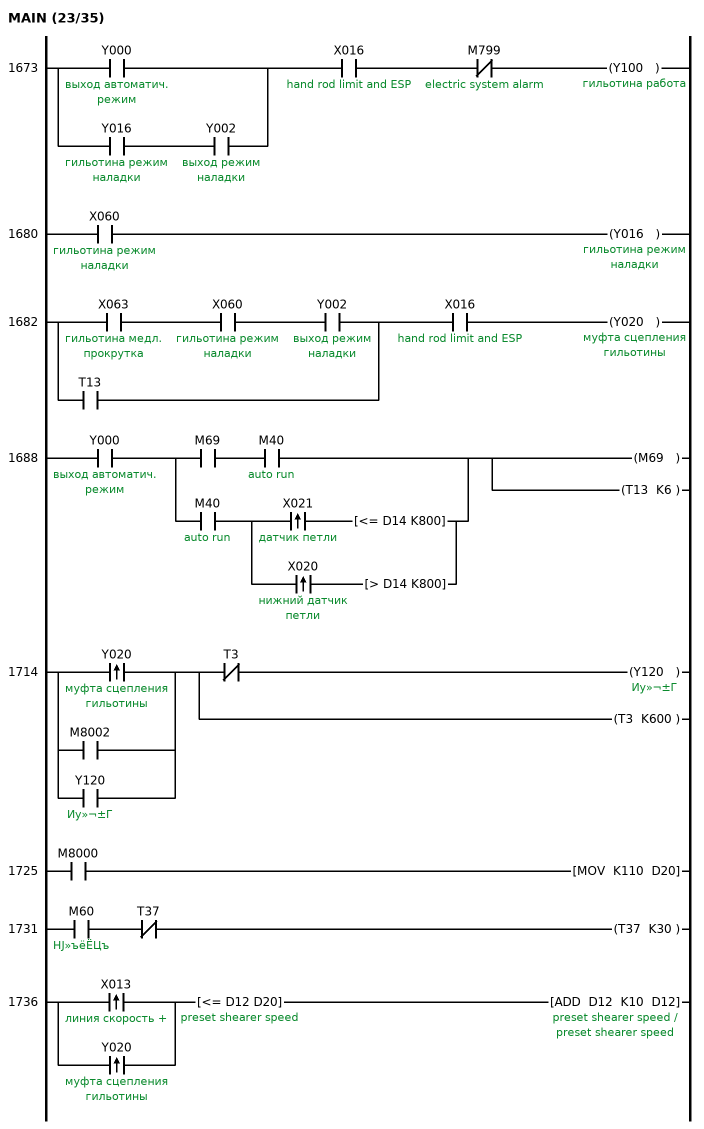
1673  LD      Y000  ; выход автоматич. режим
      LD      Y016  ; гильотина режим наладки
      AND     Y002  ; выход режим наладки
      ORB
      AND     X016  ; hand rod limit and ESP
      ANI     M799  ; electric system alarm
      OUT     Y100  ; гильотина работа
1680  LD      X060  ; гильотина режим наладки
      OUT     Y016  ; гильотина режим наладки
1682  LD      X063  ; гильотина медл. прокрутка
      AND     X060  ; гильотина режим наладки
      AND     Y002  ; выход режим наладки
      OR      T13
      AND     X016  ; hand rod limit and ESP
      OUT     Y020  ; муфта сцепления гильотины
1688  LD      Y000  ; выход автоматич. режим
      LD      M69
      AND     M40  ; auto run
      LD      M40  ; auto run
      LDP     X021  ; датчик петли
      AND<=   D14 K800
      LDP     X020  ; нижний датчик петли
      AND>    D14 K800
      ORB
      ANB
      ORB
      ANB
      OUT     M69
      OUT     T13 K6
1714  LDP     Y020  ; муфта сцепления гильотины
      OR      M8002
      OR      Y120  ; Иу»¬±Г
      MPS
      ANI     T3
      OUT     Y120  ; Иу»¬±Г
      MPP
      OUT     T3 K600
1725  LD      M8000
      MOV     K110 D20
1731  LD      M60  ; НЈ»ъёЁЦъ
      ANI     T37
      OUT     T37 K30
1736  LDP     X013  ; линия скорость +
      ORP     Y020  ; муфта сцепления гильотины
      AND<=   D12 D20  ; preset shearer speed
      ADD     D12 K10 D12
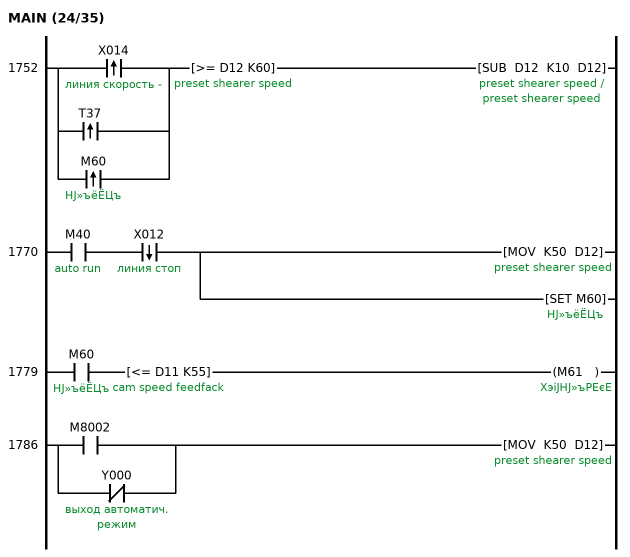
1752  LDP     X014  ; линия скорость -
      ORP     T37
      ORP     M60  ; НЈ»ъёЁЦъ
      AND>=   D12 K60  ; preset shearer speed
      SUB     D12 K10 D12
1770  LD      M40  ; auto run
      ANDF    X012  ; линия стоп
      MOV     K50 D12
      SET     M60  ; НЈ»ъёЁЦъ
1779  LD      M60  ; НЈ»ъёЁЦъ
      AND<=   D11 K55  ; cam speed feedfack
      OUT     M61  ; ХэіЈНЈ»ъРЕєЕ
1786  LD      M8002
      ORI     Y000  ; выход автоматич. режим
      MOV     K50 D12
